Staubli VAL3: getName.pgx

public program getName(string& x_sName[], num x_nIndex)
begin
  x_sName=saveData:tData[x_nIndex].name
end
